// Mitsubishi GX Works2 project: worEx02   PLC: Q02/Q02H

PROGRAM MAIN
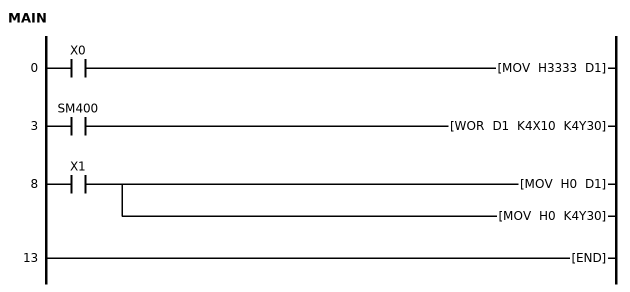
0     LD      X0
      MOV     H3333 D1
3     LD      SM400
      WOR     D1 K4X10 K4Y30
8     LD      X1
      MOV     H0 D1
      MOV     H0 K4Y30
13    END
END_PROGRAM
